(* Logix 5000 project; controller SX_V040001_C001 vendor 1 type 14 code 77 rev 16.23; software revision 16.04; part 28 of 35 *)
(* tags used below, declared in another part *)
   ALL_KINDS : INT[90];
   EMPTYING : INT[18];
   G_DInput : DINT[3];
   loading : INT[19];
   louvre : INT[11];
   NOTDOS : INT[6];
   PARAMETER : INT[501];
   T_CURRENT_EM_METER : TIMER;
   T_DELTA_EM_METER : TIMER;
   T_RPM_EM_METER : TIMER;
   T_TEMP_EM_METER : TIMER;
   TEMP : INT[14];
   TEMP_REAL : REAL[22];
(* MainProgram, continued *)

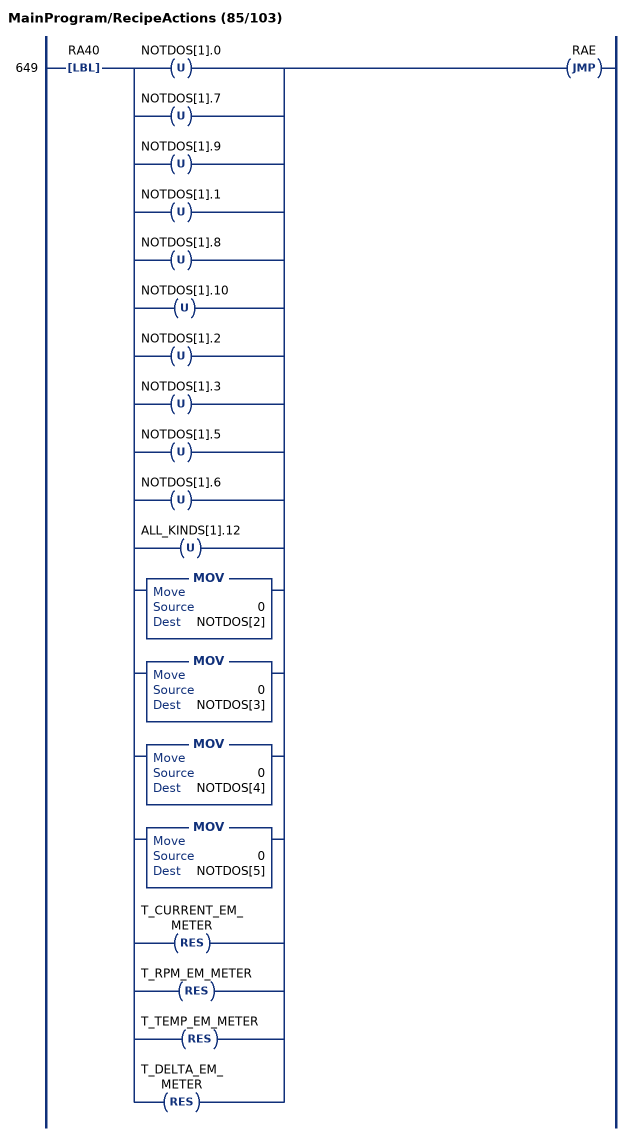
   [picture p619: MainProgram/RecipeActions rungs 649-649]
   649: LBL(RA40)[OTU(NOTDOS[1].0) ,OTU(NOTDOS[1].7) ,OTU(NOTDOS[1].9) ,OTU(NOTDOS[1].1) ,OTU(NOTDOS[1].8) ,OTU(NOTDOS[1].10) ,OTU(NOTDOS[1].2) ,OTU(NOTDOS[1].3) ,OTU(NOTDOS[1].5) ,OTU(NOTDOS[1].6) ,OTU(ALL_KINDS[1].12) ,MOV(0,NOTDOS[2]) ,MOV(0,NOTDOS[3]) ,MOV(0,NOTDOS[4]) ,MOV(0,NOTDOS[5]) ,RES(T_CURRENT_EM_METER) ,RES(T_RPM_EM_METER) ,RES(T_TEMP_EM_METER) ,RES(T_DELTA_EM_METER) ]JMP(RAE);
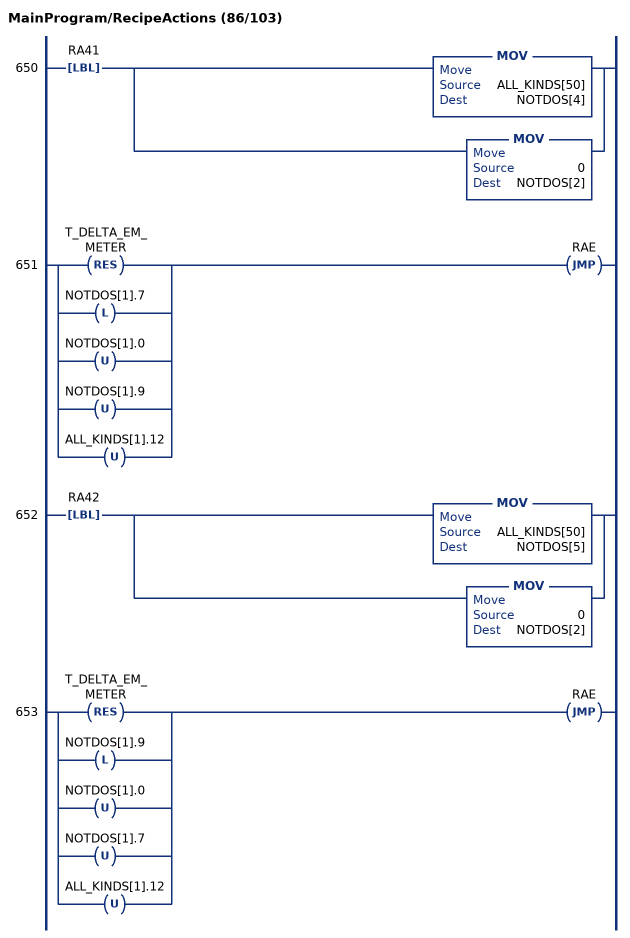
   650: LBL(RA41)[MOV(ALL_KINDS[50],NOTDOS[4]) ,MOV(0,NOTDOS[2]) ];
   651: [RES(T_DELTA_EM_METER) ,OTL(NOTDOS[1].7) ,OTU(NOTDOS[1].0) ,OTU(NOTDOS[1].9) ,OTU(ALL_KINDS[1].12) ]JMP(RAE);
   652: LBL(RA42)[MOV(ALL_KINDS[50],NOTDOS[5]) ,MOV(0,NOTDOS[2]) ];
   653: [RES(T_DELTA_EM_METER) ,OTL(NOTDOS[1].9) ,OTU(NOTDOS[1].0) ,OTU(NOTDOS[1].7) ,OTU(ALL_KINDS[1].12) ]JMP(RAE);
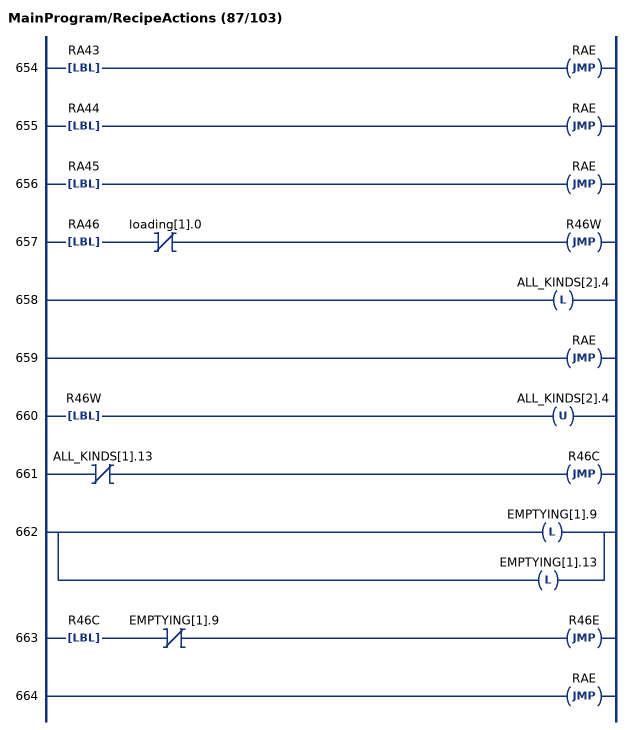
   654: LBL(RA43)JMP(RAE);
   655: LBL(RA44)JMP(RAE);
   656: LBL(RA45)JMP(RAE);
   657: LBL(RA46)XIO(loading[1].0)JMP(R46W);
   658: OTL(ALL_KINDS[2].4);
   659: JMP(RAE);
   660: LBL(R46W)OTU(ALL_KINDS[2].4);
   661: XIO(ALL_KINDS[1].13)JMP(R46C);
   662: [OTL(EMPTYING[1].9) ,OTL(EMPTYING[1].13) ];
   663: LBL(R46C)XIO(EMPTYING[1].9)JMP(R46E);
   664: JMP(RAE);
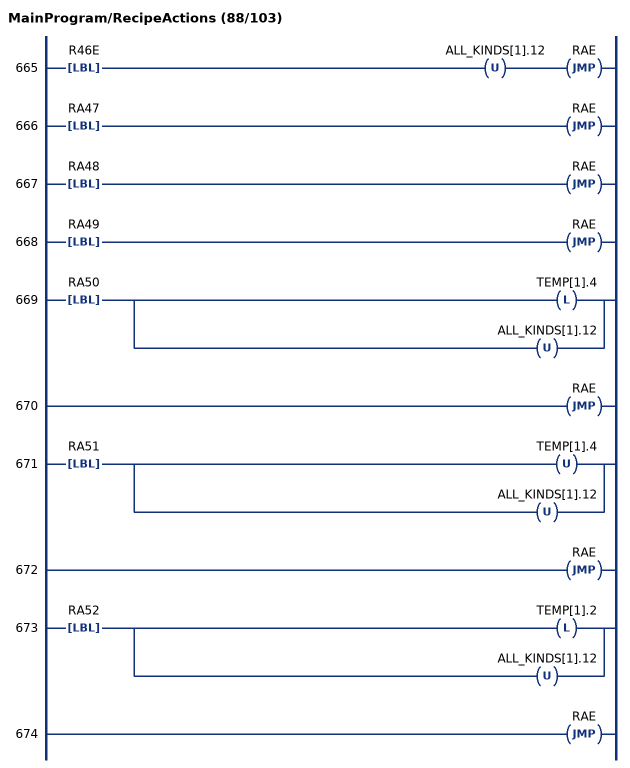
   665: LBL(R46E)OTU(ALL_KINDS[1].12)JMP(RAE);
   666: LBL(RA47)JMP(RAE);
   667: LBL(RA48)JMP(RAE);
   668: LBL(RA49)JMP(RAE);
   669: LBL(RA50)[OTL(TEMP[1].4) ,OTU(ALL_KINDS[1].12) ];
   670: JMP(RAE);
   671: LBL(RA51)[OTU(TEMP[1].4) ,OTU(ALL_KINDS[1].12) ];
   672: JMP(RAE);
   673: LBL(RA52)[OTL(TEMP[1].2) ,OTU(ALL_KINDS[1].12) ];
   674: JMP(RAE);
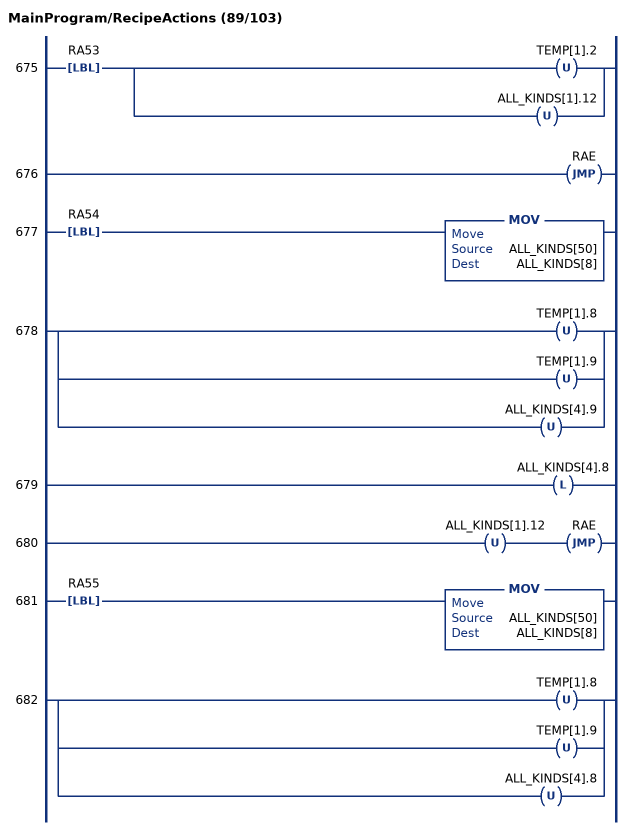
   675: LBL(RA53)[OTU(TEMP[1].2) ,OTU(ALL_KINDS[1].12) ];
   676: JMP(RAE);
   677: LBL(RA54)MOV(ALL_KINDS[50],ALL_KINDS[8]);
   678: [OTU(TEMP[1].8) ,OTU(TEMP[1].9) ,OTU(ALL_KINDS[4].9) ];
   679: OTL(ALL_KINDS[4].8);
   680: OTU(ALL_KINDS[1].12)JMP(RAE);
   681: LBL(RA55)MOV(ALL_KINDS[50],ALL_KINDS[8]);
   682: [OTU(TEMP[1].8) ,OTU(TEMP[1].9) ,OTU(ALL_KINDS[4].8) ];
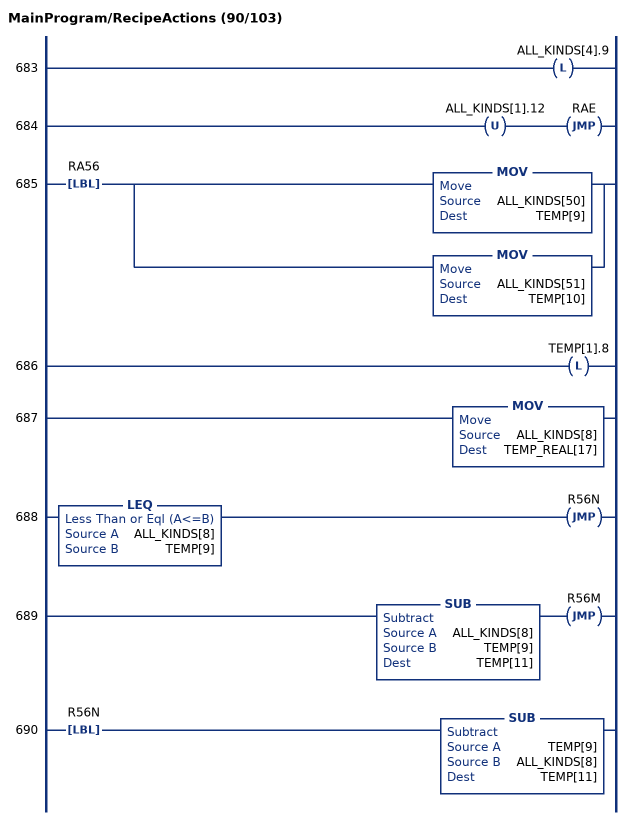
   683: OTL(ALL_KINDS[4].9);
   684: OTU(ALL_KINDS[1].12)JMP(RAE);
   685: LBL(RA56)[MOV(ALL_KINDS[50],TEMP[9]) ,MOV(ALL_KINDS[51],TEMP[10]) ];
   686: OTL(TEMP[1].8);
   687: MOV(ALL_KINDS[8],TEMP_REAL[17]);
   688: LEQ(ALL_KINDS[8],TEMP[9])JMP(R56N);
   689: SUB(ALL_KINDS[8],TEMP[9],TEMP[11])JMP(R56M);
   690: LBL(R56N)SUB(TEMP[9],ALL_KINDS[8],TEMP[11]);
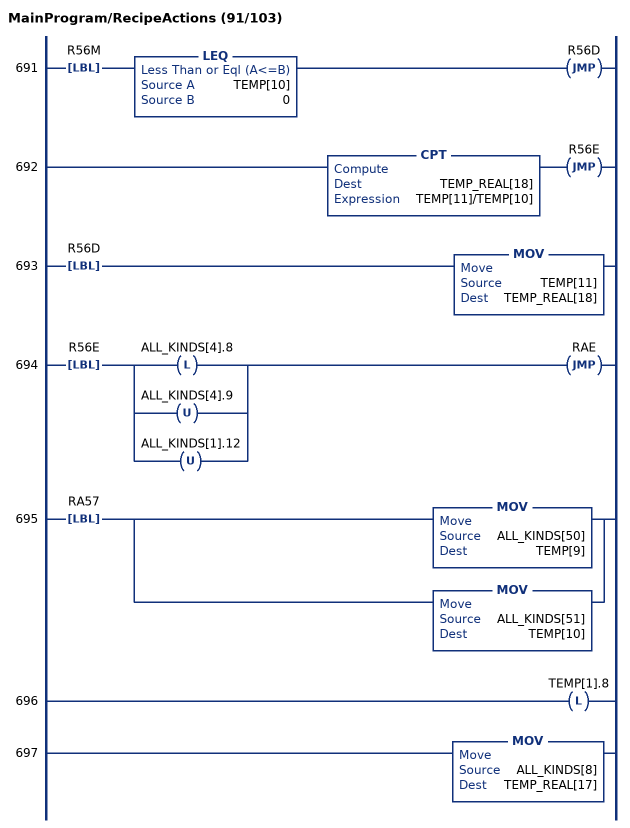
   691: LBL(R56M)LEQ(TEMP[10],0)JMP(R56D);
   692: CPT(TEMP_REAL[18],TEMP[11]/TEMP[10])JMP(R56E);
   693: LBL(R56D)MOV(TEMP[11],TEMP_REAL[18]);
   694: LBL(R56E)[OTL(ALL_KINDS[4].8) ,OTU(ALL_KINDS[4].9) ,OTU(ALL_KINDS[1].12) ]JMP(RAE);
   695: LBL(RA57)[MOV(ALL_KINDS[50],TEMP[9]) ,MOV(ALL_KINDS[51],TEMP[10]) ];
   696: OTL(TEMP[1].8);
   697: MOV(ALL_KINDS[8],TEMP_REAL[17]);
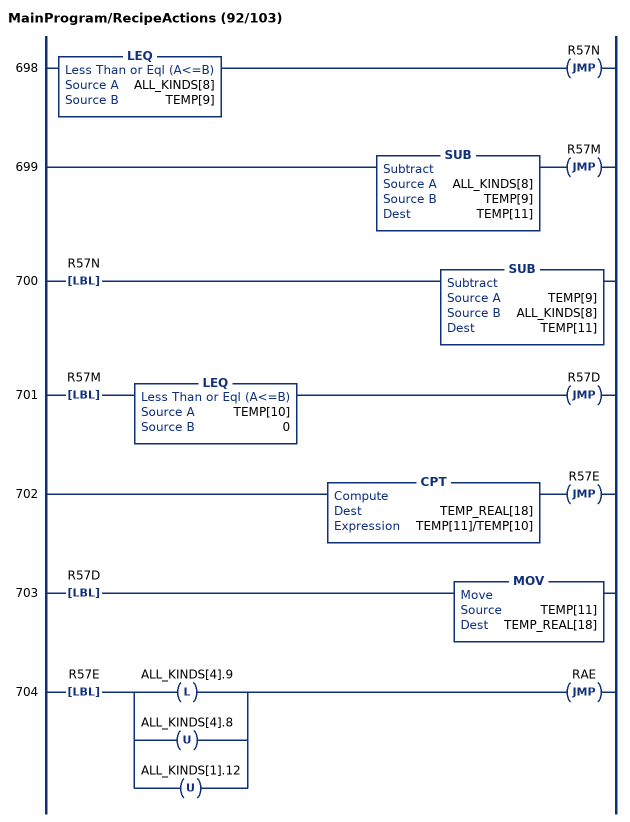
   698: LEQ(ALL_KINDS[8],TEMP[9])JMP(R57N);
   699: SUB(ALL_KINDS[8],TEMP[9],TEMP[11])JMP(R57M);
   700: LBL(R57N)SUB(TEMP[9],ALL_KINDS[8],TEMP[11]);
   701: LBL(R57M)LEQ(TEMP[10],0)JMP(R57D);
   702: CPT(TEMP_REAL[18],TEMP[11]/TEMP[10])JMP(R57E);
   703: LBL(R57D)MOV(TEMP[11],TEMP_REAL[18]);
   704: LBL(R57E)[OTL(ALL_KINDS[4].9) ,OTU(ALL_KINDS[4].8) ,OTU(ALL_KINDS[1].12) ]JMP(RAE);
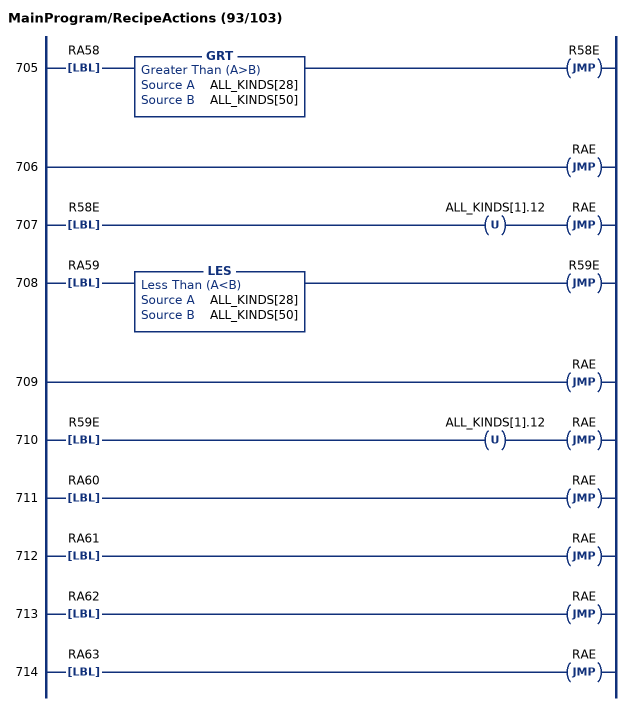
   705: LBL(RA58)GRT(ALL_KINDS[28],ALL_KINDS[50])JMP(R58E);
   706: JMP(RAE);
   707: LBL(R58E)OTU(ALL_KINDS[1].12)JMP(RAE);
   708: LBL(RA59)LES(ALL_KINDS[28],ALL_KINDS[50])JMP(R59E);
   709: JMP(RAE);
   710: LBL(R59E)OTU(ALL_KINDS[1].12)JMP(RAE);
   711: LBL(RA60)JMP(RAE);
   712: LBL(RA61)JMP(RAE);
   713: LBL(RA62)JMP(RAE);
   714: LBL(RA63)JMP(RAE);
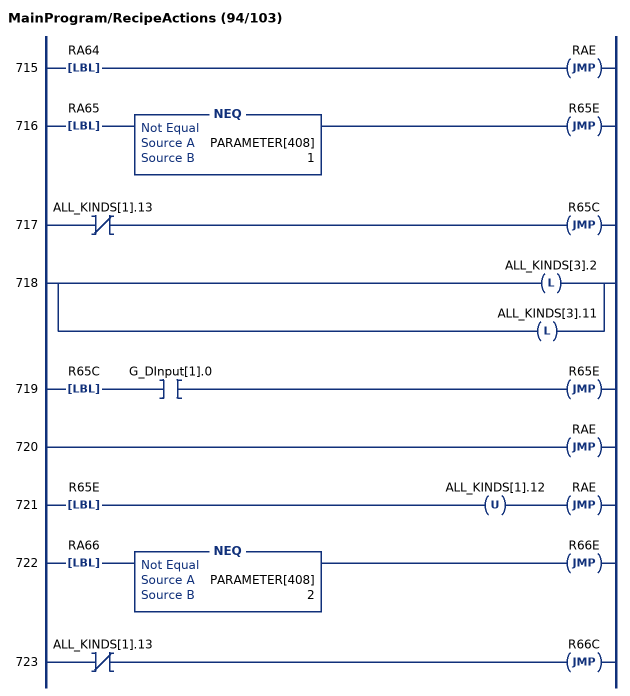
   715: LBL(RA64)JMP(RAE);
   716: LBL(RA65)NEQ(PARAMETER[408],1)JMP(R65E);
   717: XIO(ALL_KINDS[1].13)JMP(R65C);
   718: [OTL(ALL_KINDS[3].2) ,OTL(ALL_KINDS[3].11) ];
   719: LBL(R65C)XIC(G_DInput[1].0)JMP(R65E);
   720: JMP(RAE);
   721: LBL(R65E)OTU(ALL_KINDS[1].12)JMP(RAE);
   722: LBL(RA66)NEQ(PARAMETER[408],2)JMP(R66E);
   723: XIO(ALL_KINDS[1].13)JMP(R66C);
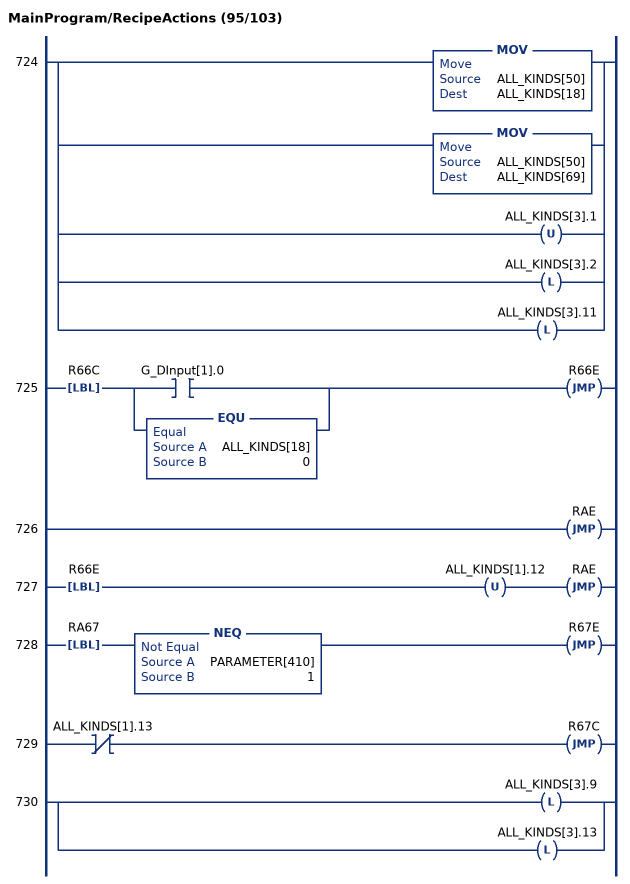
   724: [MOV(ALL_KINDS[50],ALL_KINDS[18]) ,MOV(ALL_KINDS[50],ALL_KINDS[69]) ,OTU(ALL_KINDS[3].1) ,OTL(ALL_KINDS[3].2) ,OTL(ALL_KINDS[3].11) ];
   725: LBL(R66C)[XIC(G_DInput[1].0) ,EQU(ALL_KINDS[18],0) ]JMP(R66E);
   726: JMP(RAE);
   727: LBL(R66E)OTU(ALL_KINDS[1].12)JMP(RAE);
   728: LBL(RA67)NEQ(PARAMETER[410],1)JMP(R67E);
   729: XIO(ALL_KINDS[1].13)JMP(R67C);
   730: [OTL(ALL_KINDS[3].9) ,OTL(ALL_KINDS[3].13) ];
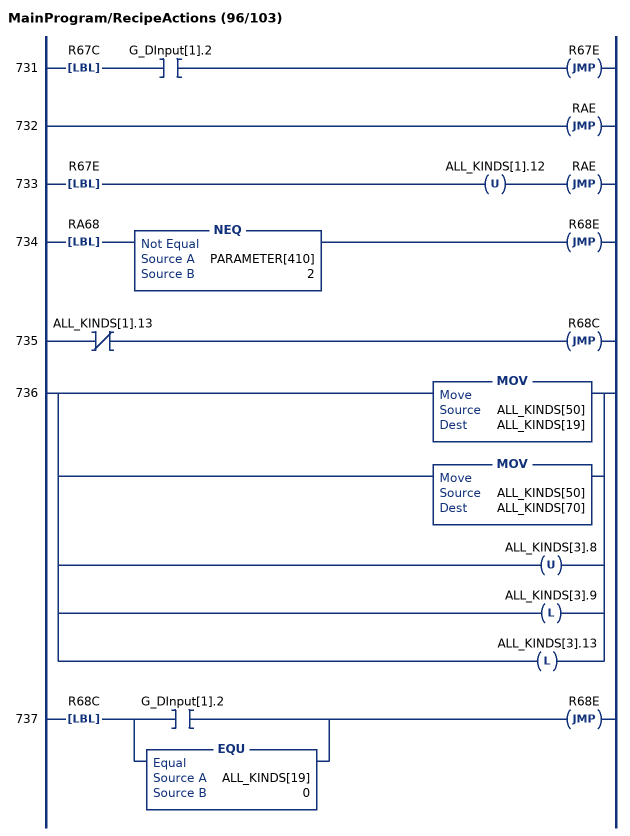
   731: LBL(R67C)XIC(G_DInput[1].2)JMP(R67E);
   732: JMP(RAE);
   733: LBL(R67E)OTU(ALL_KINDS[1].12)JMP(RAE);
   734: LBL(RA68)NEQ(PARAMETER[410],2)JMP(R68E);
   735: XIO(ALL_KINDS[1].13)JMP(R68C);
   736: [MOV(ALL_KINDS[50],ALL_KINDS[19]) ,MOV(ALL_KINDS[50],ALL_KINDS[70]) ,OTU(ALL_KINDS[3].8) ,OTL(ALL_KINDS[3].9) ,OTL(ALL_KINDS[3].13) ];
   737: LBL(R68C)[XIC(G_DInput[1].2) ,EQU(ALL_KINDS[19],0) ]JMP(R68E);
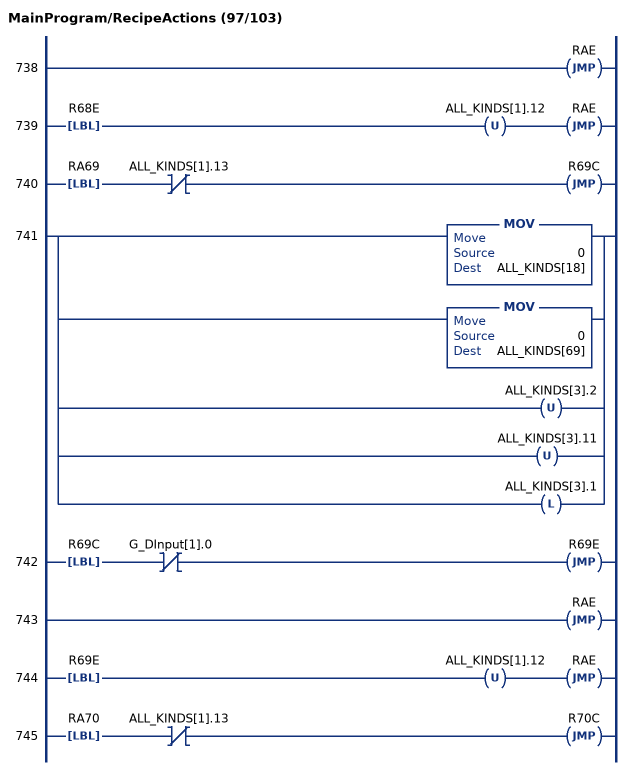
   738: JMP(RAE);
   739: LBL(R68E)OTU(ALL_KINDS[1].12)JMP(RAE);
   740: LBL(RA69)XIO(ALL_KINDS[1].13)JMP(R69C);
   741: [MOV(0,ALL_KINDS[18]) ,MOV(0,ALL_KINDS[69]) ,OTU(ALL_KINDS[3].2) ,OTU(ALL_KINDS[3].11) ,OTL(ALL_KINDS[3].1) ];
   742: LBL(R69C)XIO(G_DInput[1].0)JMP(R69E);
   743: JMP(RAE);
   744: LBL(R69E)OTU(ALL_KINDS[1].12)JMP(RAE);
   745: LBL(RA70)XIO(ALL_KINDS[1].13)JMP(R70C);
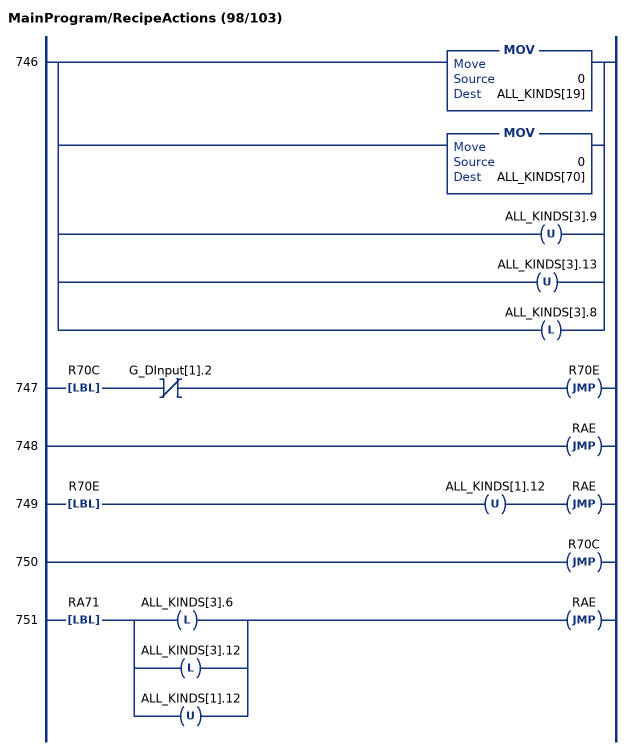
   746: [MOV(0,ALL_KINDS[19]) ,MOV(0,ALL_KINDS[70]) ,OTU(ALL_KINDS[3].9) ,OTU(ALL_KINDS[3].13) ,OTL(ALL_KINDS[3].8) ];
   747: LBL(R70C)XIO(G_DInput[1].2)JMP(R70E);
   748: JMP(RAE);
   749: LBL(R70E)OTU(ALL_KINDS[1].12)JMP(RAE);
   750: JMP(R70C);
   751: LBL(RA71)[OTL(ALL_KINDS[3].6) ,OTL(ALL_KINDS[3].12) ,OTU(ALL_KINDS[1].12) ]JMP(RAE);
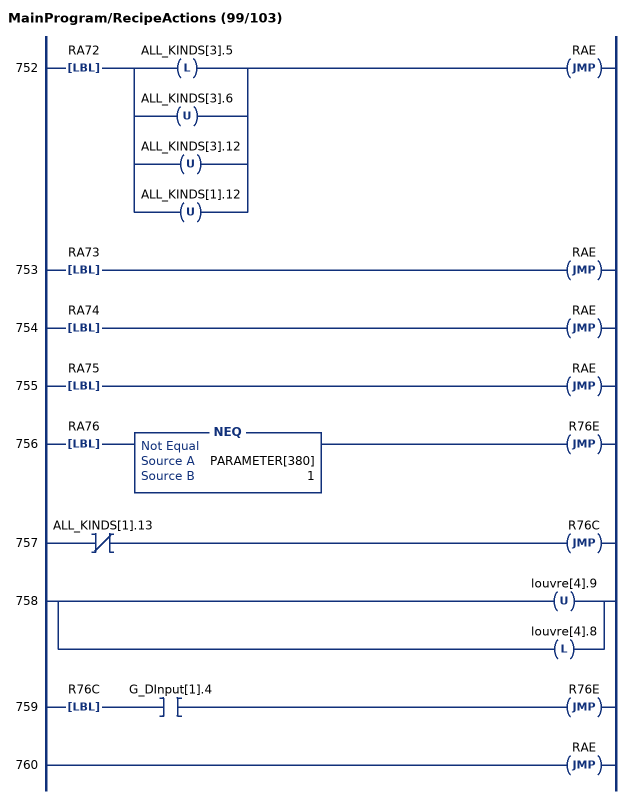
   752: LBL(RA72)[OTL(ALL_KINDS[3].5) ,OTU(ALL_KINDS[3].6) ,OTU(ALL_KINDS[3].12) ,OTU(ALL_KINDS[1].12) ]JMP(RAE);
   753: LBL(RA73)JMP(RAE);
   754: LBL(RA74)JMP(RAE);
   755: LBL(RA75)JMP(RAE);
   756: LBL(RA76)NEQ(PARAMETER[380],1)JMP(R76E);
   757: XIO(ALL_KINDS[1].13)JMP(R76C);
   758: [OTU(louvre[4].9) ,OTL(louvre[4].8) ];
   759: LBL(R76C)XIC(G_DInput[1].4)JMP(R76E);
   760: JMP(RAE);
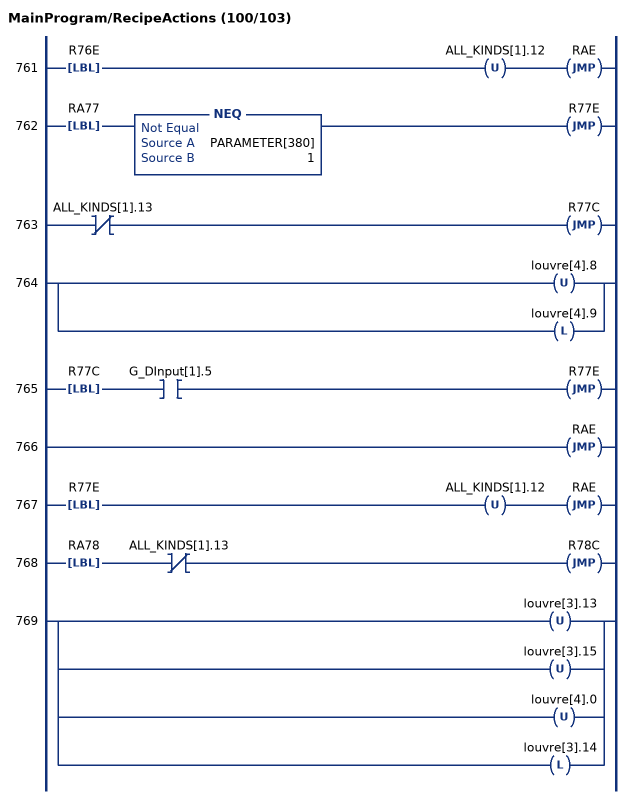
   761: LBL(R76E)OTU(ALL_KINDS[1].12)JMP(RAE);
   762: LBL(RA77)NEQ(PARAMETER[380],1)JMP(R77E);
   763: XIO(ALL_KINDS[1].13)JMP(R77C);
   764: [OTU(louvre[4].8) ,OTL(louvre[4].9) ];
   765: LBL(R77C)XIC(G_DInput[1].5)JMP(R77E);
   766: JMP(RAE);
   767: LBL(R77E)OTU(ALL_KINDS[1].12)JMP(RAE);
   768: LBL(RA78)XIO(ALL_KINDS[1].13)JMP(R78C);
   769: [OTU(louvre[3].13) ,OTU(louvre[3].15) ,OTU(louvre[4].0) ,OTL(louvre[3].14) ];
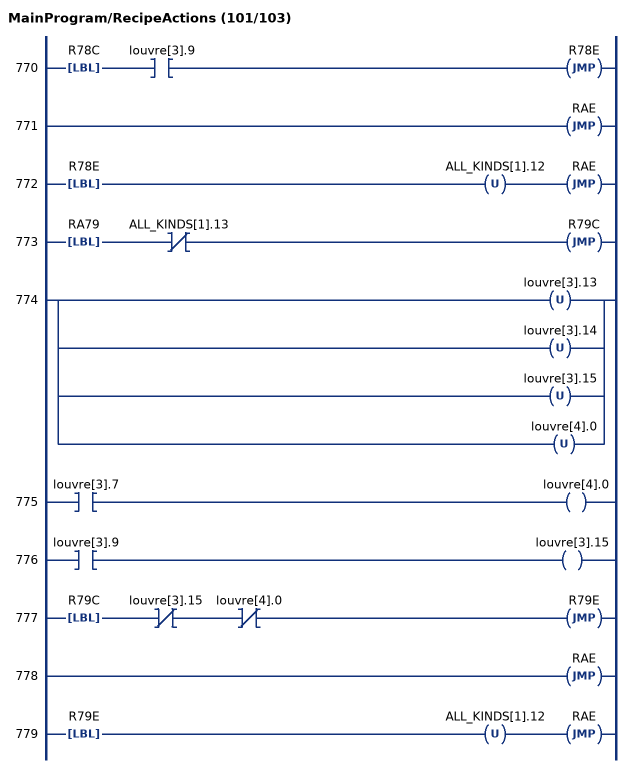
   770: LBL(R78C)XIC(louvre[3].9)JMP(R78E);
   771: JMP(RAE);
   772: LBL(R78E)OTU(ALL_KINDS[1].12)JMP(RAE);
   773: LBL(RA79)XIO(ALL_KINDS[1].13)JMP(R79C);
   774: [OTU(louvre[3].13) ,OTU(louvre[3].14) ,OTU(louvre[3].15) ,OTU(louvre[4].0) ];
   775: XIC(louvre[3].7)OTE(louvre[4].0);
   776: XIC(louvre[3].9)OTE(louvre[3].15);
   777: LBL(R79C)XIO(louvre[3].15)XIO(louvre[4].0)JMP(R79E);
   778: JMP(RAE);
   779: LBL(R79E)OTU(ALL_KINDS[1].12)JMP(RAE);
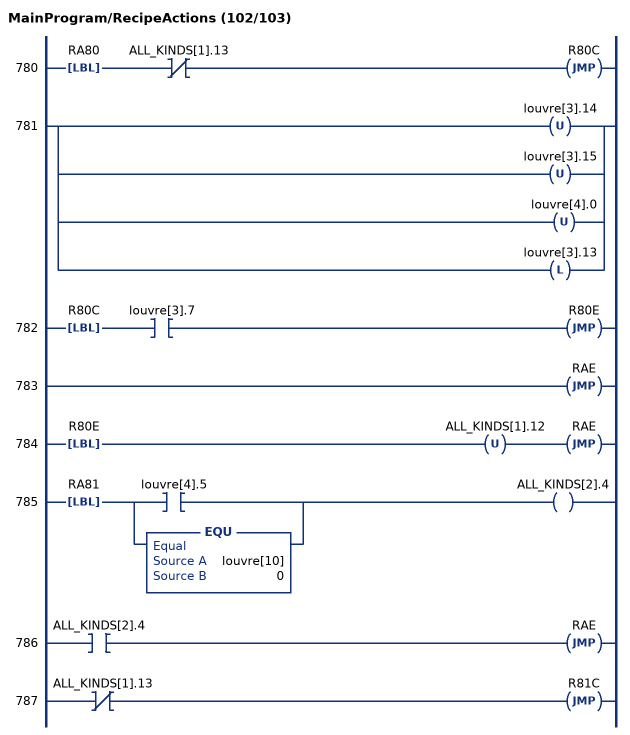
   780: LBL(RA80)XIO(ALL_KINDS[1].13)JMP(R80C);
   781: [OTU(louvre[3].14) ,OTU(louvre[3].15) ,OTU(louvre[4].0) ,OTL(louvre[3].13) ];
   782: LBL(R80C)XIC(louvre[3].7)JMP(R80E);
   783: JMP(RAE);
   784: LBL(R80E)OTU(ALL_KINDS[1].12)JMP(RAE);
   785: LBL(RA81)[XIC(louvre[4].5) ,EQU(louvre[10],0) ]OTE(ALL_KINDS[2].4);
   786: XIC(ALL_KINDS[2].4)JMP(RAE);
   787: XIO(ALL_KINDS[1].13)JMP(R81C);
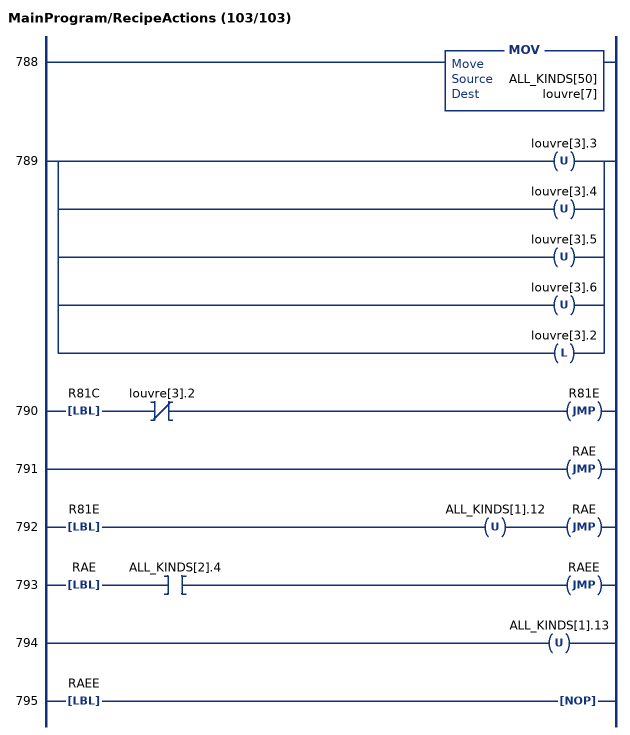
   788: MOV(ALL_KINDS[50],louvre[7]);
   789: [OTU(louvre[3].3) ,OTU(louvre[3].4) ,OTU(louvre[3].5) ,OTU(louvre[3].6) ,OTL(louvre[3].2) ];
   790: LBL(R81C)XIO(louvre[3].2)JMP(R81E);
   791: JMP(RAE);
   792: LBL(R81E)OTU(ALL_KINDS[1].12)JMP(RAE);
   793: LBL(RAE)XIC(ALL_KINDS[2].4)JMP(RAEE);
   794: OTU(ALL_KINDS[1].13);
   795: LBL(RAEE)NOP();
END_ROUTINE
